PROGRAM valve_manager
VAR
	//Repeat for each valve?
	u_3112_open_request: BOOL;
	u_3112_idle_request: BOOL;
	u_3112_cip_request: BOOL;
	u_3112_manual_request: BOOL;
	u_3112_stop_request: BOOL;
	u_3112_intlk: BOOL;
	gen_alm_active: BOOL;
	ed_routine_idle: BOOL;
	ed_routine_cip: BOOL;
	ed_routine_manual: BOOL;
	ed_routine_maint: BOOL;
	nv_3110_idle_request: BOOL;
	nv_3110_cip_request: BOOL;
	nv_3110_manual_request: BOOL;
	nv_3110_intlk: BOOL;
	nv_3110_stop_request: BOOL;
	nv_3110_open_request: BOOL;
	nv_3210_open_request: BOOL;
	nv_3310_open_request: BOOL;
	nv_3135_open_request: BOOL;
	nv_3235_open_request: BOOL;
	nv_3335_open_request: BOOL;
	nv_3372_open_request: BOOL;
	nv_3210_idle_request: BOOL;
	nv_3210_cip_request: BOOL;
	nv_3210_manual_request: BOOL;
	nv_3210_stop_request: BOOL;
	nv_3210_intlk: BOOL;
	
	nv_3310_idle_request: BOOL;
	nv_3310_cip_request: BOOL;
	nv_3310_manual_request: BOOL;
	nv_3310_stop_request: BOOL;
	nv_3310_intlk: BOOL;
	
	nv_3135_idle_request: BOOL;
	nv_3135_cip_request: BOOL;
	nv_3135_manual_request: BOOL;
	nv_3135_stop_request: BOOL;
	nv_3135_intlk: BOOL;
	
	nv_3235_idle_request: BOOL;
	nv_3235_cip_request: BOOL;
	nv_3235_manual_request: BOOL;
	nv_3235_stop_request: BOOL;
	nv_3235_intlk: BOOL;
	
	nv_3335_idle_request: BOOL;
	nv_3335_cip_request: BOOL;
	nv_3335_manual_request: BOOL;
	nv_3335_stop_request: BOOL;
	nv_3335_intlk: BOOL;
	
	nv_3372_idle_request: BOOL;
	nv_3372_cip_request: BOOL;
	nv_3372_manual_request: BOOL;
	nv_3372_stop_request: BOOL;
	nv_3372_intlk: BOOL;
	
	nv_3162_idle_request: BOOL;
	nv_3162_cip_request: BOOL;
	nv_3162_manual_request: BOOL;
	nv_3162_stop_request: BOOL;
	nv_3162_intlk: BOOL;
	nv_3162_open_request: BOOL;
	
	av_3148_idle_request: BOOL;
	av_3148_cip_request: BOOL;
	av_3148_idle_position_request: REAL;
	av_3148_position_request: REAL;
	av_3148_cip_position_request: REAL;
	av_3148_manual_position_request: REAL;
	av_3148_manual_request: BOOL;
	av_3148_maint_request: BOOL;
	av_3148_maint_position_request: REAL;
	av_3148_intlk: BOOL;
	av_3148_stop_request: BOOL;
	av_3148_open_request: BOOL;
	
	av_3248_idle_request: BOOL;
	av_3248_cip_request: BOOL;
	av_3248_idle_position_request: REAL;
	av_3248_position_request: REAL;
	av_3248_cip_position_request: REAL;
	av_3248_manual_position_request: REAL;
	av_3248_manual_request: BOOL;
	av_3248_maint_request: BOOL;
	av_3248_maint_position_request: REAL;
	av_3248_intlk: BOOL;
	av_3248_stop_request: BOOL;
	av_3248_open_request: BOOL;
	
	av_3348_idle_request: BOOL;
	av_3348_cip_request: BOOL;
	av_3348_idle_position_request: REAL;
	av_3348_position_request: REAL;
	av_3348_cip_position_request: REAL;
	av_3348_manual_position_request: REAL;
	av_3348_manual_request: BOOL;
	av_3348_maint_request: BOOL;
	av_3348_maint_position_request: REAL;
	av_3348_intlk: BOOL;
	av_3348_stop_request: BOOL;
	av_3348_open_request: BOOL;
	
END_VAR
VAR // added by the converter: edge detectors and wires of the graphical bodies
    _w1, _w2, _w3, _w4, _w5, _w6, _w7, _w8, _w9, _w10, _w11, _w12 : BOOL;
END_VAR

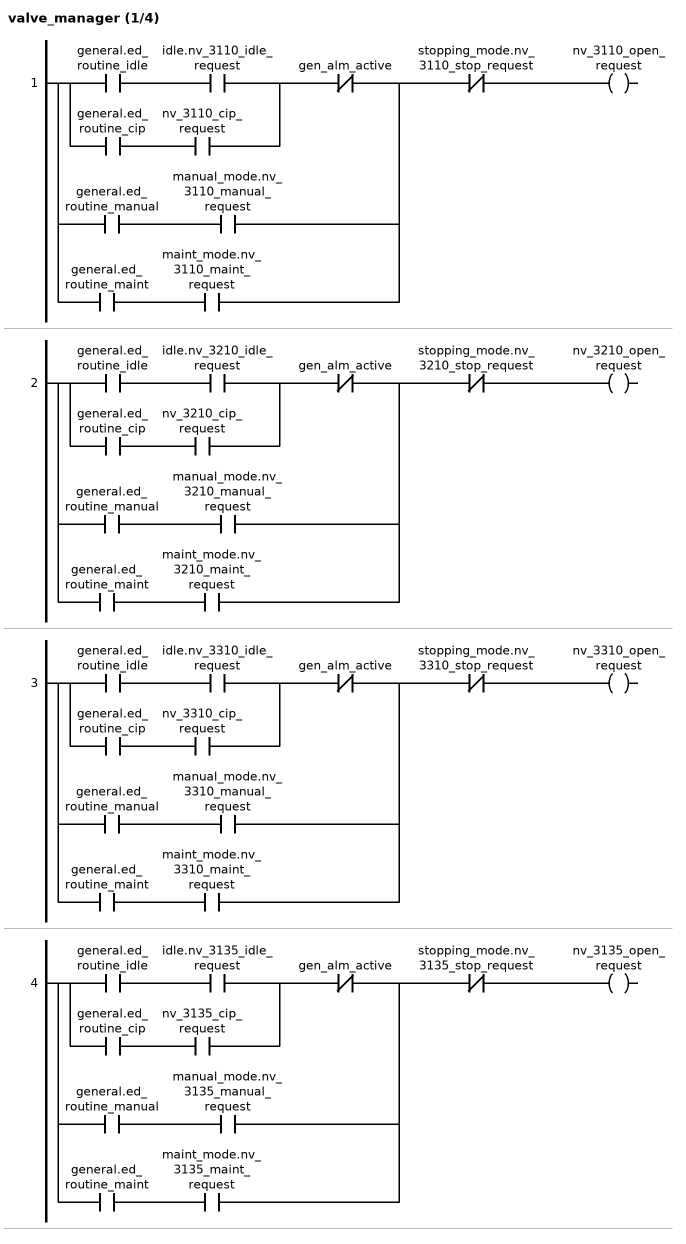
// NETWORK 1
nv_3110_open_request := ((general.ed_routine_idle AND idle.nv_3110_idle_request OR general.ed_routine_cip AND nv_3110_cip_request) AND NOT gen_alm_active OR general.ed_routine_manual AND manual_mode.nv_3110_manual_request OR general.ed_routine_maint AND maint_mode.nv_3110_maint_request) AND NOT stopping_mode.nv_3110_stop_request;

// NETWORK 2
nv_3210_open_request := ((general.ed_routine_idle AND idle.nv_3210_idle_request OR general.ed_routine_cip AND nv_3210_cip_request) AND NOT gen_alm_active OR general.ed_routine_manual AND manual_mode.nv_3210_manual_request OR general.ed_routine_maint AND maint_mode.nv_3210_maint_request) AND NOT stopping_mode.nv_3210_stop_request;

// NETWORK 3
nv_3310_open_request := ((general.ed_routine_idle AND idle.nv_3310_idle_request OR general.ed_routine_cip AND nv_3310_cip_request) AND NOT gen_alm_active OR general.ed_routine_manual AND manual_mode.nv_3310_manual_request OR general.ed_routine_maint AND maint_mode.nv_3310_maint_request) AND NOT stopping_mode.nv_3310_stop_request;

// NETWORK 4
nv_3135_open_request := ((general.ed_routine_idle AND idle.nv_3135_idle_request OR general.ed_routine_cip AND nv_3135_cip_request) AND NOT gen_alm_active OR general.ed_routine_manual AND manual_mode.nv_3135_manual_request OR general.ed_routine_maint AND maint_mode.nv_3135_maint_request) AND NOT stopping_mode.nv_3135_stop_request;

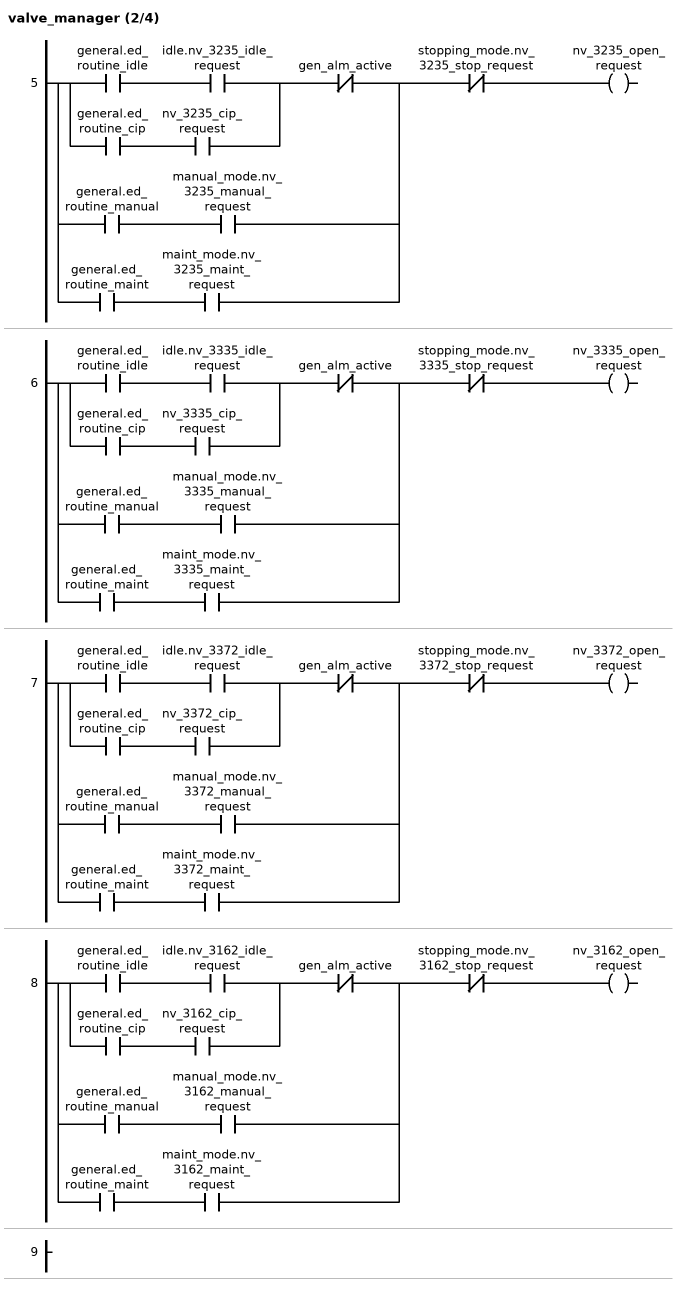
// NETWORK 5
nv_3235_open_request := ((general.ed_routine_idle AND idle.nv_3235_idle_request OR general.ed_routine_cip AND nv_3235_cip_request) AND NOT gen_alm_active OR general.ed_routine_manual AND manual_mode.nv_3235_manual_request OR general.ed_routine_maint AND maint_mode.nv_3235_maint_request) AND NOT stopping_mode.nv_3235_stop_request;

// NETWORK 6
nv_3335_open_request := ((general.ed_routine_idle AND idle.nv_3335_idle_request OR general.ed_routine_cip AND nv_3335_cip_request) AND NOT gen_alm_active OR general.ed_routine_manual AND manual_mode.nv_3335_manual_request OR general.ed_routine_maint AND maint_mode.nv_3335_maint_request) AND NOT stopping_mode.nv_3335_stop_request;

// NETWORK 7
nv_3372_open_request := ((general.ed_routine_idle AND idle.nv_3372_idle_request OR general.ed_routine_cip AND nv_3372_cip_request) AND NOT gen_alm_active OR general.ed_routine_manual AND manual_mode.nv_3372_manual_request OR general.ed_routine_maint AND maint_mode.nv_3372_maint_request) AND NOT stopping_mode.nv_3372_stop_request;

// NETWORK 8
nv_3162_open_request := ((general.ed_routine_idle AND idle.nv_3162_idle_request OR general.ed_routine_cip AND nv_3162_cip_request) AND NOT gen_alm_active OR general.ed_routine_manual AND manual_mode.nv_3162_manual_request OR general.ed_routine_maint AND maint_mode.nv_3162_maint_request) AND NOT stopping_mode.nv_3162_stop_request;

// NETWORK 9

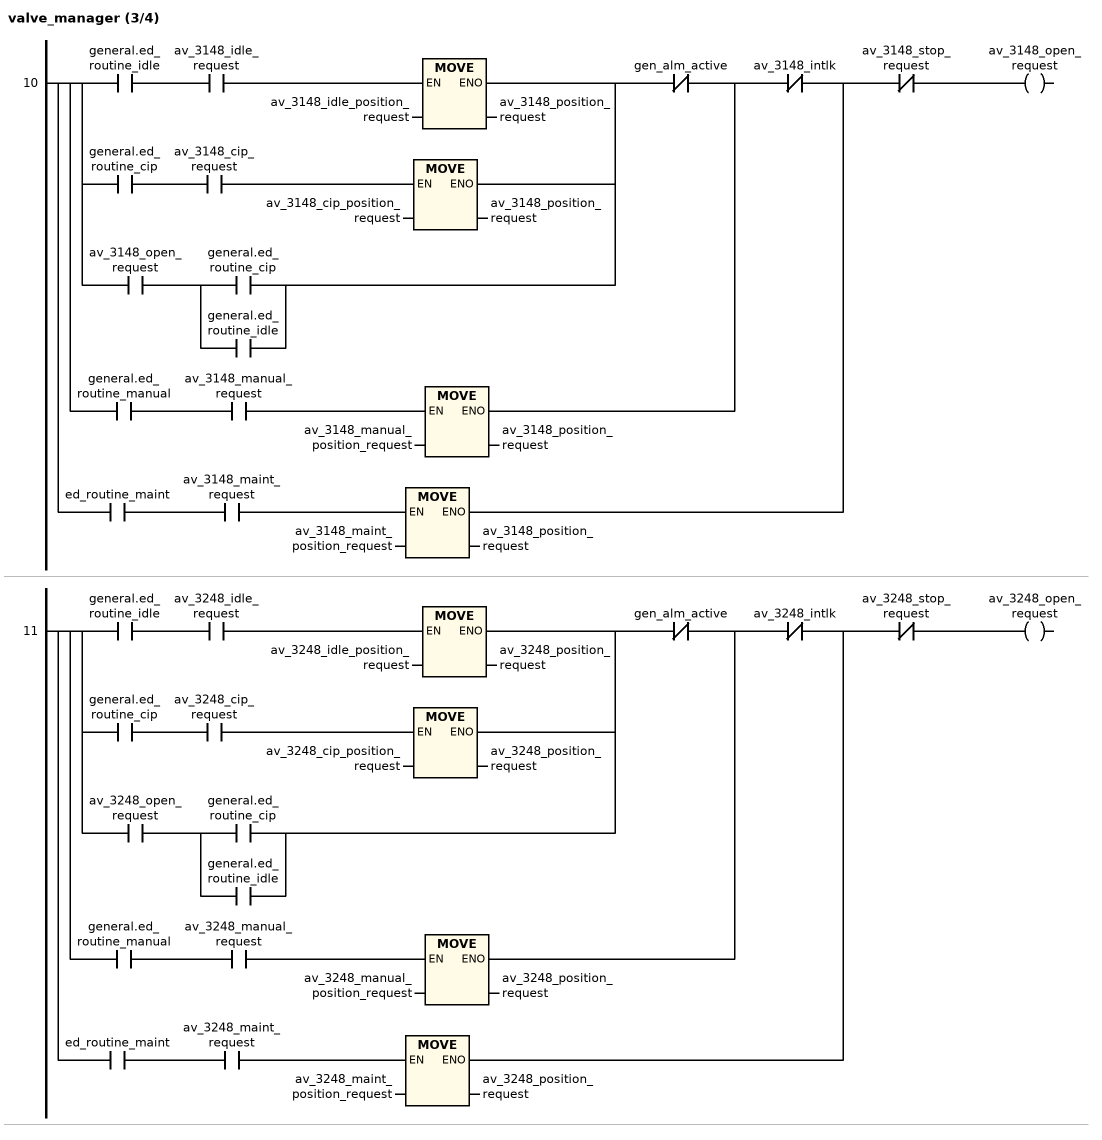
// NETWORK 10
_w1 := general.ed_routine_idle AND av_3148_idle_request;
IF _w1 THEN av_3148_position_request := av_3148_idle_position_request; END_IF
_w2 := general.ed_routine_cip AND av_3148_cip_request;
IF _w2 THEN av_3148_position_request := av_3148_cip_position_request; END_IF
_w3 := general.ed_routine_manual AND av_3148_manual_request;
IF _w3 THEN av_3148_position_request := av_3148_manual_position_request; END_IF
_w4 := ed_routine_maint AND av_3148_maint_request;
IF _w4 THEN av_3148_position_request := av_3148_maint_position_request; END_IF
av_3148_open_request := (((_w1 OR _w2 OR av_3148_open_request AND (general.ed_routine_cip OR general.ed_routine_idle)) AND NOT gen_alm_active OR _w3) AND NOT av_3148_intlk OR _w4) AND NOT av_3148_stop_request;

// NETWORK 11
_w5 := general.ed_routine_idle AND av_3248_idle_request;
IF _w5 THEN av_3248_position_request := av_3248_idle_position_request; END_IF
_w6 := general.ed_routine_cip AND av_3248_cip_request;
IF _w6 THEN av_3248_position_request := av_3248_cip_position_request; END_IF
_w7 := general.ed_routine_manual AND av_3248_manual_request;
IF _w7 THEN av_3248_position_request := av_3248_manual_position_request; END_IF
_w8 := ed_routine_maint AND av_3248_maint_request;
IF _w8 THEN av_3248_position_request := av_3248_maint_position_request; END_IF
av_3248_open_request := (((_w5 OR _w6 OR av_3248_open_request AND (general.ed_routine_cip OR general.ed_routine_idle)) AND NOT gen_alm_active OR _w7) AND NOT av_3248_intlk OR _w8) AND NOT av_3248_stop_request;

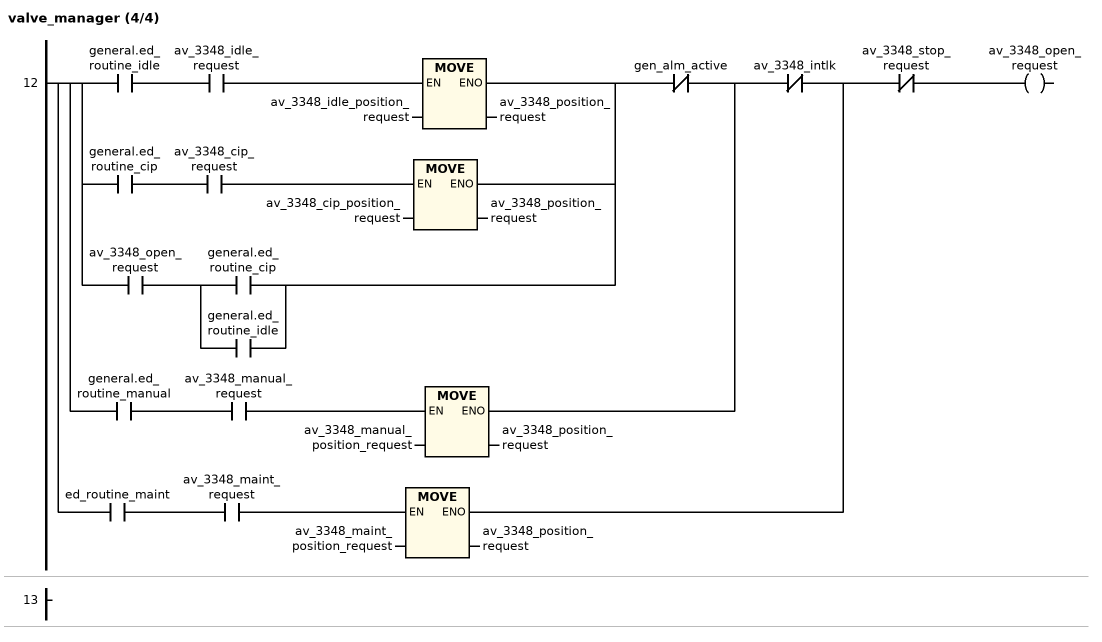
// NETWORK 12
_w9 := general.ed_routine_idle AND av_3348_idle_request;
IF _w9 THEN av_3348_position_request := av_3348_idle_position_request; END_IF
_w10 := general.ed_routine_cip AND av_3348_cip_request;
IF _w10 THEN av_3348_position_request := av_3348_cip_position_request; END_IF
_w11 := general.ed_routine_manual AND av_3348_manual_request;
IF _w11 THEN av_3348_position_request := av_3348_manual_position_request; END_IF
_w12 := ed_routine_maint AND av_3348_maint_request;
IF _w12 THEN av_3348_position_request := av_3348_maint_position_request; END_IF
av_3348_open_request := (((_w9 OR _w10 OR av_3348_open_request AND (general.ed_routine_cip OR general.ed_routine_idle)) AND NOT gen_alm_active OR _w11) AND NOT av_3348_intlk OR _w12) AND NOT av_3348_stop_request;

// NETWORK 13

END_PROGRAM

(* stored: Version 1.1.0.1, ProductVersion 3.1.4024.12
   POU valve_manager: Id {359c8254-c75f-419b-be16-97d4ba9197db}, SpecialFunc None *)
